INTERFACE I_ModuleReferenceBindings EXTENDS __SYSTEM.IQueryInterface

METHOD M_TakeOptional : I_BaseUnit
VAR_INPUT
	Name : STRING(80);
END_VAR
VAR_OUTPUT
	Present : BOOL;
	ErrorMessage : STRING(255);
END_VAR
END_METHOD

METHOD M_TakeRequired : I_BaseUnit
VAR_INPUT
	Name : STRING(80);
END_VAR
VAR_OUTPUT
	ErrorMessage : STRING(255);
END_VAR
END_METHOD

END_INTERFACE

(* stored: Version 1.1.0.1, ProductVersion 3.1.4026.18
   Itf I_ModuleReferenceBindings: Id {2a2da34d-54a3-41a2-9f99-b86c646485d1}
   Method M_TakeOptional: Id {d50f3ec8-2aec-453d-8698-8fe04702dde9}
   Method M_TakeRequired: Id {ff96cb85-1798-400c-9fcb-310cb018eeb0} *)
